// TwinCAT 3 PLC project StateMachine_Wrapper
// Title: PackML State Machine
// Company: ChrisK
// ProjectVersion: 0.0.0.1
// ProgramVersion: 3.1.4023.0
// libraries:
//   Tc2_Standard, * (Beckhoff Automation GmbH)
//   Tc2_System, * (Beckhoff Automation GmbH)
//   Tc3_Module, * (Beckhoff Automation GmbH)
//   Tc3_PackML_V2, * (Beckhoff Automation GmbH)
// project tree:
//   PackMLStateMachineWrapper/ IPmlStateMachine.TcIO, PMLStateMachine.TcPOU

// ---- PackMLStateMachineWrapper/IPmlStateMachine.TcIO
INTERFACE IPmlStateMachine

METHOD public GetCurrentMode : E_PmlProtectedUnitMode
VAR_INPUT
END_VAR
END_METHOD

METHOD GetCurrentState : E_PMLState
VAR_INPUT
END_VAR
END_METHOD

METHOD PmlModeCommand : BOOL
VAR_INPUT
	Mode : E_PMLProtectedUnitMode;
END_VAR
END_METHOD

METHOD PmlStateCommand : bool
VAR_INPUT
	Command : E_PMLCommand;
END_VAR
END_METHOD

METHOD SetStateComplete : BOOL
VAR_INPUT
END_VAR
END_METHOD

END_INTERFACE

// ---- PackMLStateMachineWrapper/PMLStateMachine.TcPOU
FUNCTION_BLOCK PMLStateMachine IMPLEMENTS IPmlStateMachine
VAR_INPUT
END_VAR
VAR_OUTPUT
END_VAR
VAR
	_pmlStateMachine : Tc3_PackML_V2.PML_StateMachine;
	_pmlModeMachine : Tc3_PackML_V2.PML_UnitModeManager;
	_subUnits : ARRAY[0..9] OF IPmlStateMachine;
	subUnitArray : ARRAY[0..9] OF ST_PMLSubUnitInfo;
	_SubUnitReference: ST_PMLSubUnitInfoRef;
	modeChangeTrigger : Tc2_Standard.R_TRIG;
	i: DINT;
END_VAR

IF _SubUnitReference.NoOfSubUnits <> 0 THEN
	FOR i := 0 TO 9 DO
		IF _subUnits[i] <> 0 THEN
			subUnitArray[i].eState := _subUnits[i].GetCurrentState();
			subUnitArray[i].Active := True;
		END_IF
	END_FOR
	_SubUnitReference.pArray := ADR(subUnitArray);
	_SubUnitReference.ArraySize := SIZEOF(subUnitArray);
END_IF

_pmlStateMachine(eMode := _pmlModeMachine.eModeStatus, stSubUnitInfoRef := _SubUnitReference);
_pmlModeMachine(eState := _pmlStateMachine.eState, bExecute := modeChangeTrigger.Q);
modeChangeTrigger();

METHOD PUBLIC GetCurrentMode : E_PmlProtectedUnitMode
VAR_INPUT
END_VAR
GetCurrentMode := _pmlModeMachine.eModeStatus;
END_METHOD

METHOD PUBLIC GetCurrentState : E_PMLState
VAR_INPUT
END_VAR
GetCurrentState := _pmlStateMachine.eState;
END_METHOD

METHOD GetNumberOfSubUnits : INT
VAR_INPUT
END_VAR
END_METHOD

METHOD PUBLIC PmlModeCommand : Bool
VAR_INPUT
	Mode : E_PMLProtectedUnitMode;
END_VAR
_pmlModeMachine.eModeCommand := Mode;
modeChangeTrigger.CLK := true;
END_METHOD

METHOD PUBLIC PmlStateCommand : BOOL
VAR_INPUT
	Command : E_PMLCommand;
END_VAR
_pmlStateMachine.eCommand := Command;
END_METHOD

METHOD PUBLIC RegisterSubUnit : BOOL
VAR_INPUT
	SubUnit : IPmlStateMachine;
END_VAR
FOR i := 0 TO 9 DO
	IF _subUnits[i] = 0 THEN
		_subUnits[i] := SubUnit;
		_SubUnitReference.NoOfSubUnits := i + 1;
		EXIT;
	END_IF
END_FOR
END_METHOD

METHOD PUBLIC SetStateComplete : BOOL
VAR_INPUT
END_VAR
_pmlStateMachine.M_StateComplete();
END_METHOD

END_FUNCTION_BLOCK
